// TIA Portal V20 export
ORGANIZATION_BLOCK "Main"   // OB1, LAD, ProgramCycle
TITLE = "Main Program Sweep (Cycle)"
{ S7_Optimized_Access := 'TRUE' }
// stored: SetENOAutomatically false
   VAR_INPUT
      Initial_Call : Bool;   // Initial call of this OB
      Remanence : Bool;   // =True, if remanent data are available
   END_VAR
BEGIN

REGION Network 1
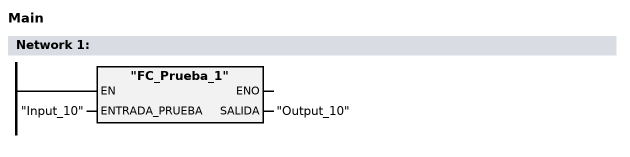
   RUNG wire#powerrail
      "FC_Prueba_1"(ENTRADA_PRUEBA := "Input_10", SALIDA => "Output_10")
   END_RUNG
   // the same network as SCL:
   "FC_Prueba_1"(ENTRADA_PRUEBA := "Input_10", SALIDA => "Output_10");
END_REGION
END_ORGANIZATION_BLOCK
